ABB RobotStudio station: tool_active_removeable_smart_modified_by_me.rsstn

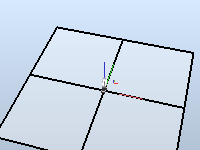
Station tool_active_removeable_smart (saved by RobotStudio format 3)
Layout (positions relative to the parent item):
  - SmartComponent_1 [smart component]
      signals: DI GripperClose, DI GripperOpen
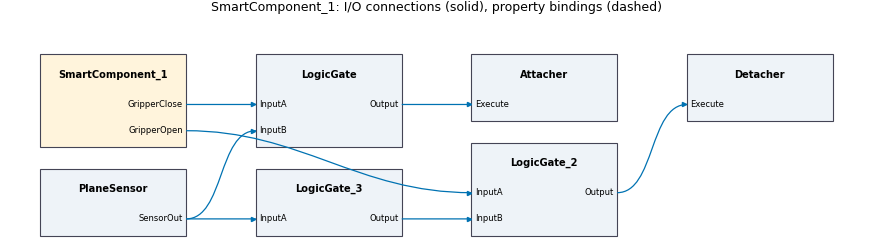
      connections:
        SmartComponent_1.GripperClose -> LogicGate.InputA
        LogicGate.Output -> Attacher.Execute
        PlaneSensor.SensorOut -> LogicGate.InputB
        SmartComponent_1.GripperOpen -> LogicGate_2.InputA
        LogicGate_2.Output -> Detacher.Execute
        PlaneSensor.SensorOut -> LogicGate_3.InputA
        LogicGate_3.Output -> LogicGate_2.InputB
    - Kosy_Tool_No_Pen [mechanism] at (0, 0, 0) mm
        TCP Kosy_Tool_No_Pen at (121, 0, 178) mm
        links: tool-m2
    - Attacher [smart component, from Components\Attacher.rslib]
        properties: Parent=Kosy_Tool_No_Pen; Flange=0; Child=Kosy_Tool_No_Pen; Mount=false; Offset=[0 0 0]; Orientation=[0 0 0]
    - Detacher [smart component, from Components\Detacher.rslib]
        properties: Child=Kosy_Tool_No_Pen; KeepPosition=true
    - PlaneSensor [smart component, from Components\PlaneSensor.rslib] at (0, -49.35, 111.88) mm, rotated rx 0 ry -89.6 rz 0 deg
        properties: Origin=[0 0 0]; Axis1=[0.1 0 0]; Axis2=[0 0.1 0]; SensedPart=(none)
      - _sensorPart_ [part, from Components\PlaneSensor.rslib]
    - LogicGate [smart component, from Components\LogicGate.rslib]
        properties: Operator=AND; Delay=0
    - LogicGate_2 [smart component, from Components\LogicGate.rslib]
        properties: Operator=AND; Delay=0
    - LogicGate_3 [smart component, from Components\LogicGate.rslib]
        properties: Operator=NOT; Delay=0
  - Frame_1 [frame] at (121, 0, 178) mm
